Fanuc KAREL source: SET_TSK_ATTR.kl

PROGRAM T
%NOLOCKGROUP
VAR
 v0 : STRING[40]
 v1 : INTEGER
 v2 : INTEGER
 v3 : INTEGER
BEGIN
 SET_TSK_ATTR(v0, v1, v2, v3)
END T
